Fanuc KAREL source: ko00059.KL

PROGRAM KO00059
%STACKSIZE=65535
%PRIORITY=65535
%NOLOCKGROUP
VAR
P1 : XYZWPR
P2 : XYZWPREXT
F : BOOLEAN
OUT : XYZWPREXT
BEGIN
F=TRUE
-- UNSAFE_SOURCE_IR line 11: OUT = MIRROR(convert_xyzwpr_to_xyzwprext(P1), convert_xyzwprext_to_position(P2), F)
END KO00059
